FUNCTION_BLOCK UA_ObserverIds (* OPC UA node IDs of the published state variables, below UaRoot *)
  (* Standard: 61499-2 *)
  (* Version 2.0, 2026-09-27, Project contributors, Filling cell reference model *)
  PACKAGE fillingcell;
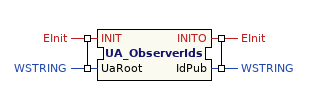
  EVENT_INPUT
    INIT : EInit WITH UaRoot;
  END_EVENT
  EVENT_OUTPUT
    INITO : EInit WITH IdPub;
  END_EVENT
  VAR_INPUT
    UaRoot : WSTRING;
  END_VAR
  VAR_OUTPUT
    IdPub : WSTRING;
  END_VAR
  EC_STATES
    INIT : INIT -> INITO;
  END_STATES
  ALGORITHM INIT IN ST:
IdPub := CONCAT(CONCAT(CONCAT(CONCAT(CONCAT(CONCAT(CONCAT(CONCAT(CONCAT(CONCAT(CONCAT(CONCAT(CONCAT(CONCAT(CONCAT(CONCAT(CONCAT(CONCAT("opc_ua[WRITE;", UaRoot), "/State/NeedleUp;"), UaRoot), "/State/NeedleDown;"), UaRoot), "/State/VialPresent;"), UaRoot), "/State/FilledMl;"), UaRoot), "/State/Stoppered;"), UaRoot), "/State/Checked;"), UaRoot), "/State/DoorClosed;"), UaRoot), "/State/Valid;"), UaRoot), "/State/Safe]");
  END_ALGORITHM
END_FUNCTION_BLOCK
